(*
/*
 *****************************************************************************
 * timeUTCToMJD: convert struct ccsTIMEVAL into modified Julian date
 *
 *  IN   ut: time in UT
 *  OUT    : Modified julian date 
 ***************************************************************************** 
 */
*)
FUNCTION F_timeUTCToMJD : LREAL
VAR_INPUT
	ut:	T_TIMEVAL;
END_VAR
VAR
	mjd:	LREAL;
END_VAR

(*
DOUBLE timeUTCToMJD(vltTIMEVAL *ut)   /* time in UT                       */
    {
    DOUBLE mjd;                       /* modified julian date             */
   /*
    *# Get Julian Date from UT 
    */
    mjd = timeUTCToJD(ut);
    
   /*
    *# Convert Julian Date into Modified Julian Date according to the formula:
    *# MJD = JD - 2400000.5;
    */
    mjd-= CONST3;
    return(mjd);    
    }
*)

// Get Julian Date from UT 
mjd := F_timeUTCToJD(ut);

(*
*# Convert Julian Date into Modified Julian Date according to the formula:
*# MJD = JD - 2400000.5;
*)
F_timeUTCToMJD	:= mjd - GCL.C_CONST3;

END_FUNCTION

(* stored: Version 1.1.0.1, ProductVersion 3.1.4022.9
   POU F_timeUTCToMJD: Id {b04e8dea-84be-4e6f-a443-dbf392717c45}, SpecialFunc None *)
